RoboDK station: Set-Up.rdk

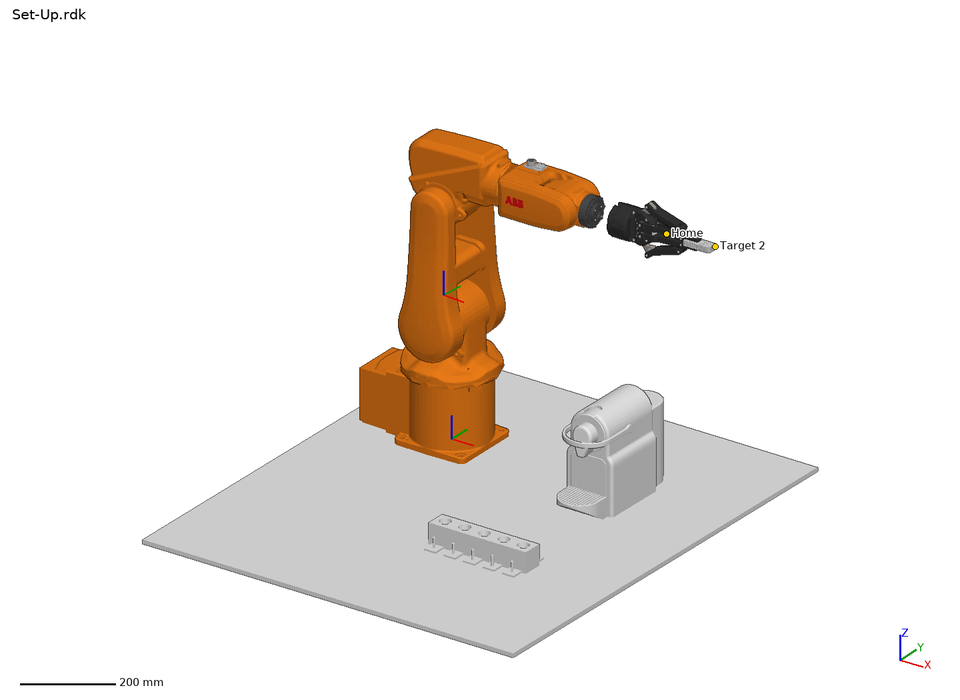
[picture v0: the station drawn from its stored meshes, robots at their saved joint values, targets as dots, program paths as lines]
Station Set-Up (saved by RoboDK 5.6.7). Poses are relative to the parent item; angles as X-Y-Z fixed-axis rotations.
Station parameters (name, value as stored): LIN64
  - frame ABB IRB 120-3/0.6 Base at (-2.05, 0, 0) mm
    - robot ABB IRB 120-3/0.6: 6 axes, payload 3 kg, reach 580 mm, repeatability 0.01 mm, weight 25 kg
        modified DH rows (alpha deg, a mm, theta deg, d mm): 0, 0, 0, 290; -90, 0, -90, 0; 0, 270, 0, 0; -90, 70, 0, 302; 90, 0, 0, 0; -90, 0, 180, 72
        joint limits [-165, -110, -90, -160, -120, -400] to [165, 110, 70, 160, 120, 400]; home [0, 0, 0, 0, 0, 0]; saved at [0, 0, 0, 0, 0, 0]
      - tool RobotiQ 2F-140 Gripper (Closed), TCP at (0, 0, 290) mm, size 124 x 75 x 244.3 mm
    - frame Frame 3 at (-574.7, 791.46, -141.86) mm, rotated rx -0.23 ry -0.22 rz -4.88 deg
      - object scene setup no arms part STL orientated at (300, 0, 0) mm, rotated rx 90 ry 0 rz 0 deg, size 1033.7 x 286 x 1171.5 mm, geometry from scene setup no arms part STL orientated.STL
      - target Home (joint target) at (1189.1, -696.14, 764.61) mm, rotated rx 129.14 ry 89.69 rz 134.02 deg; joints [0, -5.412, 5.183, 0.001, 0.228, -0.002] of ABB IRB 120-3/0.6
      - target Target 2 (Cartesian target) at (1304.43, -676.29, 764.21) mm, rotated rx 129.14 ry 89.69 rz 134.02 deg; joints [1.884, 0.213, -0.207, 89.804, -1.883, -89.803] of ABB IRB 120-3/0.6
  - program Prog1 (3 instructions, listed below)

--- program Prog1 (robot ABB IRB 120-3/0.6) ---
  Set Ref.: Frame 3
  Set Tool: RobotiQ 2F-140 Gripper (Closed)
  MoveJ (Home)
